(* CODESYS project FanucSimpleLibrary.library
   Author: Yonatan Avrakh
   Version: 0.1.0.0
   Description: A simple library allowing fast integration with FANUC robot
   Title: FanucSimple
   DefaultNamespace: FanucSimple
   Placeholder: FanucSimple
   Company: Beckhoff Automation IL

Project tree, tasks and I/O mapping:
  libraries: Tc2_Standard, * (Beckhoff Automation GmbH); Tc2_System, * (Beckhoff Automation GmbH)
  DUTs/
    data type E_FanucCstopiState
    data type E_FanucEnableState
    data type E_FanucFaultResetState
    data type E_FanucHomingState
    data type E_FanucStartProgramState
    data type ST_FanucControl
    data type ST_FanucStatus
  GVLs/
  POUs/
    function block FB_FanucControl [ST]
    function block FB_FanucCycleStop [ST]
    function block FB_FanucEnable [ST]
    function block FB_FanucFaultReset [ST]
    function block FB_FanucHoming [ST]
    function block FB_FanucOverwrite [ST]
    function block FB_FanucStartProgram [ST]
    function block FB_FanucStatus [ST]
  Version/
    global variables Global_Version
  VISUs/
*)

// DUTs/E_FanucCstopiState
(*
  States for FB_FanucCycleStop.
  Sequence: Idle → Pulsing → Done (→ Idle)
*)
TYPE E_FanucCstopiState :
(
	Idle    := 0,   // Waiting for bTrigger rising edge.
	Pulsing := 1,   // CSTOPI signal pulsed for 20 ms.
	Done    := 2    // Cycle stop complete – bDone TRUE for one scan, then → Idle.
);
END_TYPE

// DUTs/E_FanucEnableState
(*
  States for FB_FanucEnable.
  The enable sequence progresses: Idle → ClearFault → CheckTP → WaitReady → Ready.
  From Ready, conditions are monitored continuously (priority order):
    bFault             → ClearFault
    bTP_Enabled        → CheckTP
    bExtIMSTP = FALSE  → EmergencyStop (E-stop; resumes via ClearFault when released)
    bExtSFSPD = FALSE  → SafeSpeed     (fence open; robot at safe speed; bReady FALSE)
    bExtHold  = FALSE  → Paused        (HOLD only drops; IMSTP/SFSPD/ENBL held)
  Toggle bEnable FALSE→TRUE to retry from Idle after an Error.
*)
TYPE E_FanucEnableState :
(
  Idle              := 0,   // Waiting for bEnable. ENBL de-asserted; bExt* signals pass through.
  ClearFault        := 1,   // Assert Fault_Reset pulse until bFault clears (5 s timeout → Error).
  CheckTP           := 3,   // Wait for bTP_Enabled = FALSE (operator must switch TP off).
  WaitReady         := 4,   // Wait for bCmd_Enabled AND bSystem_Ready (5 s timeout → Error).
  Ready             := 5,   // Robot is ready. Monitor for all safety/fault conditions.
  Paused            := 6,   // bExtHold = FALSE: HOLD dropped, IMSTP/SFSPD/ENBL held. Resumes when bExtHold TRUE.
  EmergencyStop     := 7,   // bExtIMSTP = FALSE: E-stop active. ENBL held. Resumes via ClearFault when IMSTP released.
  SafeSpeed         := 8,   // bExtSFSPD = FALSE: fence open, robot at safe speed. bReady FALSE. Resumes when fence closes.
  Error             := 99   // Enable sequence failed. ENBL de-asserted. Toggle bEnable to reset.
);
END_TYPE

// DUTs/E_FanucFaultResetState
(*
  States for FB_FanucFaultReset.
  Sequence: Idle → SendPulse → WaitClear → Done (→ Idle).
  Error on timeout; reset by setting bReset FALSE.
*)
TYPE E_FanucFaultResetState :
(
  Idle      := 0,   // Waiting for bReset rising edge.
  SendPulse := 1,   // FAULT_RESET signal pulsed for 20 ms (robot acts on rising edge).
  WaitClear := 2,   // Waiting for bFault = FALSE (configurable timeout → Error).
  Done      := 3,   // Fault cleared – bDone TRUE for one scan, then → Idle.
  Error     := 99   // Fault persisted after reset attempt. Set bReset FALSE to reset.
);
END_TYPE

// DUTs/E_FanucHomingState
(*
  States for FB_FanucHoming.
  Sequence: Idle → RequestHome → WaitComplete → Done (→ Idle).
  Error on timeout; reset by setting bStart FALSE.
*)
TYPE E_FanucHomingState :
(
  Idle         := 0,   // Waiting for bStart rising edge (interlocked by bReady).
  RequestHome  := 1,   // HOME signal (UI[7]) pulsed for 20 ms to trigger homing macro.
  WaitComplete := 2,   // Waiting for bAt_Home (UO[7]) = TRUE (configurable timeout).
  Done         := 3,   // Homing confirmed – bDone TRUE for one scan, then → Idle.
  Error        := 99   // Timeout waiting for completion. Set bStart FALSE to reset.
);
END_TYPE

// DUTs/E_FanucStartProgramState
(*
  States for FB_FanucStartProgram.
  Sequence: Idle → Pulsing → Done (→ Idle)
  Error on invalid program number; reset by setting bStart FALSE.
*)
TYPE E_FanucStartProgramState :
(
	Idle    := 0,   // Waiting for bStart rising edge.
	Pulsing := 1,   // Program start bits asserted for 200 ms.
	Done    := 2,   // Pulse complete – bDone TRUE for one scan, then → Idle.
	Error   := 99   // Program number out of range. Set bStart FALSE to reset.
);
END_TYPE

// DUTs/ST_FanucControl
TYPE ST_FanucControl : STRUCT
//  Control byte 0
  IMSTP        :  BOOL;  //  (* bit 0 *)
  Hold        :  BOOL;  //  (* bit 1 *)
  SFSPD        :  BOOL;  //  (* bit 2 *)
  Cycle_stop      :  BOOL;  //  (* bit 3 *)
  Fault_Reset      :  BOOL;  //  (* bit 4 *)
  Start        :  BOOL;  //  (* bit 5 *)
  Home        :  BOOL;  //  (* bit 6 *)
  Enable        :  BOOL;  //  (* bit 7 *)

//  Control byte 1  (UI[9..16]  RSR1..RSR8 / PNS1..PNS8)
  Start_Program1    :  BOOL;  //  UI[9]  RSR1 / PNS bit 0
  Start_Program2    :  BOOL;  //  UI[10] RSR2 / PNS bit 1
  Start_Program3    :  BOOL;  //  UI[11] RSR3 / PNS bit 2
  Start_Program4    :  BOOL;  //  UI[12] RSR4 / PNS bit 3
  Start_Program5    :  BOOL;  //  UI[13] RSR5 / PNS bit 4
  Start_Program6    :  BOOL;  //  UI[14] RSR6 / PNS bit 5
  Start_Program7    :  BOOL;  //  UI[15] RSR7 / PNS bit 6
  Start_Program8    :  BOOL;  //  UI[16] RSR8 / PNS bit 7

//  Control byte 2  (UI[17..18])
  PNS_Strobe      :  BOOL;
  Prod_Start      :  BOOL;  //  UI[18] PROD_START – triggers PNS program execution

//  Control byte 3  (GI[25..33] – user-defined output)
  Overwrite            :  BYTE;
END_STRUCT
END_TYPE

// DUTs/ST_FanucStatus
TYPE ST_FanucStatus : STRUCT
  //DI[0,0] - Status Byte 0
  bCmd_Enabled  : BOOL;  (* bit 0 *)
  bSystem_Ready  : BOOL;  (* bit 1 *)
  bPrg_Running  : BOOL;  (* bit 2 *)
  bPrg_Paused    : BOOL;  (* bit 3 *)
  bMotion_Held  : BOOL;  (* bit 4 *)
  bFault      : BOOL;  (* bit 5 *)
  bAt_Home    : BOOL;  (* bit 6 *)
  bTP_Enabled    : BOOL;  (* BIT 7 *)

  //DI[0,1] - Status Byte 1
  bBatteryAlarm :BOOL; (* bit 1 *)
  bBusy :BOOL;  (* bit 2 *)

  //DI[0,2] - Status Byte 2
  bProg_Start1ACK  : BOOL;  (* bit 1 *)
  bProg_Start2ACK  : BOOL;  (* bit 2 *)
  bProg_Start3ACK  : BOOL;  (* bit 3 *)
  bProg_Start4ACK  : BOOL;  (* bit 4 *)
  bProg_Start5ACK  : BOOL;  (* bit 5 *)
  bProg_Start6ACK  : BOOL;  (* bit 6 *)
  bProg_Start7ACK  : BOOL;  (* bit 7 *)
  bProg_Start8ACK  : BOOL;  (* bit 8 *)

END_STRUCT
END_TYPE

// Version/Global_Version
{attribute 'TcGenerated'}
{attribute 'no-analysis'}
{attribute 'linkalways'}
// This function has been automatically generated from the project information.
VAR_GLOBAL CONSTANT
	{attribute 'const_non_replaced'}
	stLibVersion_FanucSimple : ST_LibVersion := (iMajor := 0, iMinor := 1, iBuild := 0, iRevision := 0, nFlags := 1, sVersion := '0.1.0.0');
END_VAR

// POUs/FB_FanucControl
(* Writes ST_FanucControl fields TO EtherCAT output bytes (aDO). Call every scan AFTER all control logic is complete. Pass GVL_Fanuc.DO0 AT the call site
*)
FUNCTION_BLOCK FB_FanucControl
VAR_IN_OUT
  aDO : ARRAY[0..15] OF BYTE; // Injected EtherCAT output array – pass GVL_Fanuc.DO0
END_VAR
VAR_INPUT
  stControl : ST_FanucControl;
END_VAR


// Control Byte 0  (aDO[0])  —  UI[1..8]
aDO[0].0 := stControl.IMSTP;        // UI[1]  *IMSTP       NC – hold TRUE; FALSE = software E-stop
aDO[0].1 := stControl.Hold;         // UI[2]  *HOLD        NC – hold TRUE; FALSE = decelerate & pause
aDO[0].2 := stControl.SFSPD;        // UI[3]  *SFSPD       NC – hold TRUE; FALSE = safe-speed limit
aDO[0].3 := stControl.Cycle_stop;   // UI[4]  CSTOPI       pulse to stop/abort current cycle
aDO[0].4 := stControl.Fault_Reset;  // UI[5]  FAULT_RESET  pulse to reset clearable alarms
aDO[0].5 := stControl.Start;        // UI[6]  START        falling-edge resumes paused program
aDO[0].6 := stControl.Home;         // UI[7]  HOME         macro use only
aDO[0].7 := stControl.Enable;       // UI[8]  ENBL         NC – hold TRUE; FALSE = disable all motion

// Control Byte 1  (aDO[1])  —  UI[9..16]  RSR / PNS
aDO[1].0 := stControl.Start_Program1; // UI[9]  RSR1 / PNS bit 0
aDO[1].1 := stControl.Start_Program2; // UI[10] RSR2 / PNS bit 1
aDO[1].2 := stControl.Start_Program3; // UI[11] RSR3 / PNS bit 2
aDO[1].3 := stControl.Start_Program4; // UI[12] RSR4 / PNS bit 3
aDO[1].4 := stControl.Start_Program5; // UI[13] RSR5 / PNS bit 4
aDO[1].5 := stControl.Start_Program6; // UI[14] RSR6 / PNS bit 5
aDO[1].6 := stControl.Start_Program7; // UI[15] RSR7 / PNS bit 6
aDO[1].7 := stControl.Start_Program8; // UI[16] RSR8 / PNS bit 7

// Control Byte 2  (aDO[2])  —  UI[17..18]
aDO[2].0 := stControl.PNS_Strobe;                   // UI[17] reserved
aDO[2].1 := stControl.Prod_Start;   // UI[18] PROD_START – triggers PNS program execution

// Control Byte 3  (aDO[3])  —  GI[25..33] user-defined output
aDO[3] := stControl.Overwrite;

END_FUNCTION_BLOCK

// POUs/FB_FanucCycleStop
// Sends the CSTOPI (UI[4]) Cycle Stop signal to the FANUC robot.
// Rising edge on bTrigger sends a 20 ms pulse; bDone goes TRUE for one scan when complete.
FUNCTION_BLOCK FB_FanucCycleStop
VAR_INPUT
  bTrigger   : BOOL;   // Rising edge: send Cycle Stop command
END_VAR
VAR_IN_OUT
  stControl  : ST_FanucControl;   // Control struct – wire same instance as FB_FanucEnable output
END_VAR
VAR_OUTPUT
  bBusy      : BOOL;               // TRUE while pulse is active
  bDone      : BOOL;               // One scan TRUE when cycle stop pulse is complete
  eState     : E_FanucCstopiState; // Current state (diagnostic / HMI)
END_VAR
VAR
  _eState   : E_FanucCstopiState := E_FanucCstopiState.Idle;
  rtTrigger : R_TRIG;
  tonPulse  : TON;   // 20 ms CSTOPI pulse width
END_VAR
VAR CONSTANT
  tPulse : TIME := T#20MS;   // CSTOPI minimum pulse width (spec: ≥15 ms)
END_VAR

(*
  FB_FanucCycleStop
  Sends a 20 ms CSTOPI pulse (UI[4]) to the FANUC robot.

  CSTOPI clears programs waiting on RSR. The effect on the running program depends
  on the "CSTOPI for ABORT" setting on the controller (MENU → SYSTEM → Config item 6):
    DISABLE – program stops at the end of its current cycle (graceful stop).
    ENABLE  – program is immediately aborted at the current line.
  This FB sends the pulse unconditionally; the controller setting determines the behaviour.

  Usage:
    - Call every PLC cycle.
    - Pass the same stControl instance used by FB_FanucEnable and FB_FanucControl.
    - Give bTrigger a rising edge to issue the command.
    - bDone goes TRUE for one scan when the 20 ms pulse is complete.
*)

// ---------- Edge detect ----------
rtTrigger(CLK := bTrigger);

// ---------- State machine ----------
CASE _eState OF

  E_FanucCstopiState.Idle:
    stControl.Cycle_stop := FALSE;
    tonPulse(IN := FALSE);
    IF rtTrigger.Q THEN
      _eState := E_FanucCstopiState.Pulsing;
    END_IF

  E_FanucCstopiState.Pulsing:
    // Assert CSTOPI for 20 ms, then → Done.
    tonPulse(IN := TRUE, PT := tPulse);
    stControl.Cycle_stop := NOT tonPulse.Q;  // TRUE for first 20 ms, then FALSE
    IF tonPulse.Q THEN
      stControl.Cycle_stop := FALSE;
      tonPulse(IN := FALSE);
      _eState := E_FanucCstopiState.Done;
    END_IF

  E_FanucCstopiState.Done:
    // bDone is TRUE for one scan (derived below), then → Idle.
    stControl.Cycle_stop := FALSE;
    _eState := E_FanucCstopiState.Idle;

ELSE
  _eState := E_FanucCstopiState.Idle;

END_CASE

// ---------- Derived outputs ----------
eState := _eState;
bBusy  := (_eState = E_FanucCstopiState.Pulsing);
bDone  := (_eState = E_FanucCstopiState.Done);

END_FUNCTION_BLOCK

// POUs/FB_FanucEnable
// Runs the FANUC enable sequence (IMSTP/HOLD/SFSPD → ClearFault → CheckTP → WaitReady → Ready).
// Validates interlock preconditions before enabling. Set bEnable TRUE to start; toggle FALSE→TRUE to reset after error.
FUNCTION_BLOCK FB_FanucEnable
VAR_INPUT
  bEnable    : BOOL;           // Command: TRUE to run enable sequence
  stStatus   : ST_FanucStatus; // Live robot status (from FB_FanucStatus)
  // External interlock signals – Normally Closed convention: TRUE = normal, FALSE = activate stop/hold
  // May be driven by HMI, safety PLC, or TwinCAT logic. Merged at the call site; this FB sees one value per signal.
  bExtIMSTP  : BOOL;  // External *IMSTP: FALSE = E-stop requested
  bExtHold   : BOOL;  // External *HOLD:  FALSE = pause/hold requested
  bExtSFSPD  : BOOL;  // External *SFSPD: FALSE = safe-speed limit requested
  bExtStart  : BOOL;  // External Start command: rising edge triggers a 20 ms START pulse (Ready state only)
END_VAR
VAR_OUTPUT
  bReady          : BOOL;                // Robot is ready to execute programs
  bError          : BOOL;                // Enable sequence failed – check eState
  bTPWarning      : BOOL;                // TP switch is ON – operator action needed
  eState          : E_FanucEnableState;  // Current state (diagnostic / HMI)
  stControl       : ST_FanucControl;     // Control outputs – wire to FB_FanucControl
END_VAR
VAR
  _eState          : E_FanucEnableState := E_FanucEnableState.Idle;
  tonReadyTimeout  : TON;   // Timeout waiting for CMDENBL + SYSRDY (5 s → Error)
  rtExtStart       : R_TRIG;  // Rising-edge detector for bExtStart
  tonStartPulse    : TON;   // 20 ms START pulse generator
END_VAR
VAR CONSTANT
  tStartPulse : TIME := T#20MS;  // START signal minimum pulse width
END_VAR

(*
  FB_FanucEnable
  Implements the FANUC robot enable sequence as a state machine.

  Sequence (per FANUC UI/UO signal spec):
    0. Idle       – bEnable must be TRUE and all interlocks in required state before proceeding.
    1. ClearFault – Waits for bFault = FALSE. Does NOT send a reset pulse; use FB_FanucFaultReset.
    2. CheckTP    – Wait for bTP_Enabled = FALSE. TP switch must be OFF for remote control.
    3. WaitReady  – Wait for bCmd_Enabled AND bSystem_Ready (5 s timeout → Error).
    4. Ready      – bReady = TRUE. Continuously monitors for fault/TP/hold/interlock changes.

  To reset after Error: set bEnable FALSE, then TRUE again.

  Fault clearing:
    This FB does not send FAULT_RESET. When in ClearFault state, call FB_FanucFaultReset
    (passing the same stControl instance) and trigger it with bReset. FB_FanucEnable will
    transition out of ClearFault automatically once bFault = FALSE.

  NC signal behaviour (Option A – passive when disabled):
    When bEnable = FALSE (Idle or Error): IMSTP, HOLD, SFSPD are held TRUE (non-asserting).
    ENBL = FALSE is the primary gate; additional stop assertions would cause unnecessary alarms.
    When in any active state: NC signals reflect bExt* inputs directly.

  Emergency Stop (bExtIMSTP = FALSE from Ready/Paused/SafeSpeed):
    → EmergencyStop. NC signal drops immediately; robot stops. ENBL stays asserted for recovery.
    No fault-clear while IMSTP is low. When bExtIMSTP returns TRUE → ClearFault.

  Safe Speed (bExtSFSPD = FALSE from Ready/Paused):
    → SafeSpeed. Robot continues at safe speed; bReady = FALSE.
    When bExtSFSPD returns TRUE: → Ready (if bExtHold TRUE) or → Paused.

  Pause / Hold (bExtHold = FALSE from Ready):
    → Paused. Only HOLD is dropped; IMSTP, SFSPD and ENBL remain asserted.
    When bExtHold returns TRUE → Ready.

  Start (bExtStart):
    Rising edge in Ready state triggers a 20 ms pulse on stControl.Start (UI[6]).
    Must be FALSE before the enable sequence can begin.

  Library usage:
    - Call every PLC cycle.
    - Pass fbStatus.stStatus into stStatus.
    - Wire stControl output to FB_FanucControl (inject aDO at call site).
    - Program start, homing, and cycle-stop bits are not managed here;
      handle those in the calling application or a dedicated FB.
*)

// ------------------- NC safety signals — always reflect external inputs directly -------------------
stControl.IMSTP := bExtIMSTP;
stControl.Hold  := bExtHold;
stControl.SFSPD := bExtSFSPD;

// ------------------- State machine – transition logic only -------------------
CASE _eState OF

  E_FanucEnableState.Idle:
    tonReadyTimeout(IN := FALSE);
    // All interlock preconditions must be met before starting the enable sequence.
    IF bEnable AND bExtIMSTP AND bExtHold AND bExtSFSPD AND NOT bExtStart THEN
      _eState := E_FanucEnableState.ClearFault;
    END_IF

  E_FanucEnableState.ClearFault:
    // Wait for bFault to clear. No pulse is sent here – use FB_FanucFaultReset for that.
    // Abort back to Idle if bEnable dropped or any interlock was lost mid-sequence.
    IF NOT bEnable OR NOT bExtIMSTP OR NOT bExtHold OR NOT bExtSFSPD THEN
      _eState := E_FanucEnableState.Idle;
    ELSIF NOT stStatus.bFault THEN
      _eState := E_FanucEnableState.CheckTP;
    END_IF

  E_FanucEnableState.CheckTP:
    // bTPWarning is derived below; stay here until operator switches TP off.
    // Abort if bEnable dropped or any interlock was lost mid-sequence.
    IF NOT bEnable OR NOT bExtIMSTP OR NOT bExtHold OR NOT bExtSFSPD THEN
      _eState := E_FanucEnableState.Idle;
    ELSIF NOT stStatus.bTP_Enabled THEN
      tonReadyTimeout(IN := FALSE);
      _eState := E_FanucEnableState.WaitReady;
    END_IF

  E_FanucEnableState.WaitReady:
    // Wait for CMDENBL (UO1) and SYSRDY (UO2) to confirm the robot is ready.
    // Interlock loss takes highest priority – abort cleanly rather than time out.
    tonReadyTimeout(IN := TRUE, PT := T#5S);
    IF NOT bEnable OR NOT bExtIMSTP OR NOT bExtHold OR NOT bExtSFSPD THEN
      tonReadyTimeout(IN := FALSE);
      _eState := E_FanucEnableState.Idle;
    ELSIF stStatus.bCmd_Enabled AND stStatus.bSystem_Ready THEN
      tonReadyTimeout(IN := FALSE);
      _eState := E_FanucEnableState.Ready;
    ELSIF stStatus.bTP_Enabled THEN
      tonReadyTimeout(IN := FALSE);
      _eState := E_FanucEnableState.CheckTP;
    ELSIF stStatus.bFault THEN
      tonReadyTimeout(IN := FALSE);
      _eState := E_FanucEnableState.ClearFault;
    ELSIF tonReadyTimeout.Q THEN
      _eState := E_FanucEnableState.Error;
    END_IF

  E_FanucEnableState.Ready:
    // Monitor all conditions (priority: fault > TP > E-stop > SafeSpeed > Hold).
    IF NOT bEnable THEN
      _eState := E_FanucEnableState.Idle;
    ELSIF stStatus.bFault THEN
      _eState := E_FanucEnableState.ClearFault;
    ELSIF stStatus.bTP_Enabled THEN
      _eState := E_FanucEnableState.CheckTP;
    ELSIF NOT bExtIMSTP THEN
      _eState := E_FanucEnableState.EmergencyStop;
    ELSIF NOT bExtSFSPD THEN
      _eState := E_FanucEnableState.SafeSpeed;
    ELSIF stStatus.bMotion_Held THEN
      _eState := E_FanucEnableState.Paused;
    END_IF

  E_FanucEnableState.Paused:
    // HOLD NC already low via passthrough. ENBL remains asserted.
    IF NOT bEnable THEN
      _eState := E_FanucEnableState.Idle;
    ELSIF stStatus.bFault THEN
      _eState := E_FanucEnableState.ClearFault;
    ELSIF stStatus.bTP_Enabled THEN
      _eState := E_FanucEnableState.CheckTP;
    ELSIF NOT bExtIMSTP THEN
      _eState := E_FanucEnableState.EmergencyStop;
    ELSIF NOT bExtSFSPD THEN
      _eState := E_FanucEnableState.SafeSpeed;
    ELSIF NOT stStatus.bMotion_Held THEN
      _eState := E_FanucEnableState.Ready;
    END_IF

  E_FanucEnableState.EmergencyStop:
    // IMSTP NC already low via passthrough. ENBL stays asserted for recovery.
    // Do NOT attempt fault-clear while IMSTP is still low.
    IF NOT bEnable THEN
      _eState := E_FanucEnableState.Idle;
    ELSIF stStatus.bTP_Enabled THEN
      _eState := E_FanucEnableState.CheckTP;
    ELSIF bExtIMSTP THEN
      // E-stop released – robot almost certainly alarmed; pass through ClearFault.
      _eState := E_FanucEnableState.ClearFault;
    END_IF

  E_FanucEnableState.SafeSpeed:
    // SFSPD NC already low via passthrough; robot runs at safe speed.
    IF NOT bEnable THEN
      _eState := E_FanucEnableState.Idle;
    ELSIF stStatus.bFault THEN
      _eState := E_FanucEnableState.ClearFault;
    ELSIF stStatus.bTP_Enabled THEN
      _eState := E_FanucEnableState.CheckTP;
    ELSIF NOT bExtIMSTP THEN
      _eState := E_FanucEnableState.EmergencyStop;
    ELSIF bExtSFSPD THEN
      // Fence closed – resume; honour hold state.
      IF bExtHold THEN
        _eState := E_FanucEnableState.Ready;
      ELSE
        _eState := E_FanucEnableState.Paused;
      END_IF
    END_IF

  E_FanucEnableState.Error:
    // ENBL de-asserted (derived below). Reset by toggling bEnable FALSE → TRUE.
    IF NOT bEnable THEN
      tonReadyTimeout(IN := FALSE);
      _eState := E_FanucEnableState.Idle;
    END_IF

ELSE
  _eState := E_FanucEnableState.Error;

END_CASE

//-------------------START pulse-------------------
//  Convert rising edge of bExtStart into a clean 20 ms pulse on stControl.Start.
//  Gated by Ready state – rising edges in any other state are ignored.
//  If we leave Ready mid-pulse (e.g. fault occurs), the timer resets cleanly. *)
rtExtStart(CLK := bExtStart AND (_eState = E_FanucEnableState.Ready));
tonStartPulse(IN := tonStartPulse.IN OR rtExtStart.Q, PT := tStartPulse);
IF tonStartPulse.Q THEN
  tonStartPulse(IN := FALSE);
END_IF
IF _eState <> E_FanucEnableState.Ready THEN
  tonStartPulse(IN := FALSE);
END_IF

// -------------------Derived outputs-------------------
// Evaluated after the state machine so they always reflect the current state. *)
eState             := _eState;
stControl.Enable   := (_eState <> E_FanucEnableState.Idle)  AND (_eState <> E_FanucEnableState.Error);
stControl.Start    := (_eState =  E_FanucEnableState.Ready) AND tonStartPulse.IN;
bReady             := (_eState =  E_FanucEnableState.Ready);
bError             := (_eState =  E_FanucEnableState.Error);
bTPWarning         := (_eState =  E_FanucEnableState.CheckTP) AND stStatus.bTP_Enabled;

END_FUNCTION_BLOCK

// POUs/FB_FanucFaultReset
// Sends a FAULT_RESET pulse to the FANUC robot and waits for the fault to clear.
// Trigger with a rising edge on bReset. Toggle bReset FALSE to reset after Error.
FUNCTION_BLOCK FB_FanucFaultReset
VAR_INPUT
  bReset   : BOOL;            // Rising edge: send fault reset pulse to robot
  stStatus : ST_FanucStatus;  // Live robot status (from FB_FanucStatus)
END_VAR
VAR_IN_OUT
  stControl : ST_FanucControl;  // Control struct – pass same instance as FB_FanucEnable.stControl
END_VAR
VAR_OUTPUT
  bBusy  : BOOL;                    // TRUE while reset sequence is in progress
  bDone  : BOOL;                    // One scan TRUE when fault is confirmed cleared
  bError : BOOL;                    // Fault persisted after reset – operator action needed
  eState : E_FanucFaultResetState;  // Current state (diagnostic / HMI)
END_VAR
VAR
  _eState    : E_FanucFaultResetState := E_FanucFaultResetState.Idle;
  rtReset    : R_TRIG;
  tonPulse   : TON;  // 20 ms FAULT_RESET pulse
  tonTimeout : TON;  // Timeout waiting for fault to clear after reset
END_VAR
VAR CONSTANT
  tResetPulse   : TIME := T#20MS;  // FAULT_RESET minimum pulse width
  tFaultTimeout : TIME := T#5S;    // Max time to wait for fault to clear after reset
END_VAR

(*
  FB_FanucFaultReset
  Sends a timed FAULT_RESET pulse (UI[5]) to the robot and monitors bFault until clear.

  Sequence:
    1. SendPulse  – Assert FAULT_RESET for 20 ms. Robot acts on the rising edge.
    2. WaitClear  – Wait for bFault (UO[4]) = FALSE. Timeout → Error.
    3. Done       – bDone TRUE for one scan, then → Idle.

  Usage:
    - Call every PLC cycle.
    - Pass the same stControl instance used by FB_FanucEnable (VAR_IN_OUT, by reference).
    - Trigger with a rising edge on bReset (e.g. HMI button, or automatic from application logic).
    - Check bDone for one-scan confirmation that the fault cleared.
    - Check bError if the fault did not clear; set bReset FALSE to reset.

  Relationship with FB_FanucEnable:
    - FB_FanucEnable.ClearFault state waits for bFault = FALSE without sending any pulse.
    - This FB is responsible for the actual reset signal; the application decides when to trigger it.
    - Typically called when FB_FanucEnable.eState = ClearFault and the operator requests a reset.
*)

rtReset(CLK := bReset);

CASE _eState OF

  E_FanucFaultResetState.Idle:
    stControl.Fault_Reset := FALSE;
    tonPulse(IN := FALSE);
    tonTimeout(IN := FALSE);
    IF rtReset.Q THEN
      _eState := E_FanucFaultResetState.SendPulse;
    END_IF

  E_FanucFaultResetState.SendPulse:
    // Assert FAULT_RESET for exactly 20 ms. Robot acts on the rising edge.
    tonPulse(IN := TRUE, PT := tResetPulse);
    stControl.Fault_Reset := NOT tonPulse.Q; // TRUE for first 20 ms, then FALSE
    IF tonPulse.Q THEN
      stControl.Fault_Reset := FALSE;
      tonPulse(IN := FALSE);
      _eState := E_FanucFaultResetState.WaitClear;
    END_IF

  E_FanucFaultResetState.WaitClear:
    // Pulse complete; wait for robot to confirm the fault is gone.
    stControl.Fault_Reset := FALSE;
    tonTimeout(IN := TRUE, PT := tFaultTimeout);
    IF NOT stStatus.bFault THEN
      tonTimeout(IN := FALSE);
      _eState := E_FanucFaultResetState.Done;
    ELSIF tonTimeout.Q THEN
      _eState := E_FanucFaultResetState.Error;
    END_IF

  E_FanucFaultResetState.Done:
    // bDone is TRUE for exactly one scan (derived below), then return to Idle.
    stControl.Fault_Reset := FALSE;
    _eState := E_FanucFaultResetState.Idle;

  E_FanucFaultResetState.Error:
    // Fault did not clear after reset. Reset this FB by setting bReset FALSE.
    stControl.Fault_Reset := FALSE;
    IF NOT bReset THEN
      tonPulse(IN := FALSE);
      tonTimeout(IN := FALSE);
      _eState := E_FanucFaultResetState.Idle;
    END_IF

ELSE
  _eState := E_FanucFaultResetState.Error;

END_CASE

// ---------- Derived outputs ---------- *)
eState := _eState;
bBusy  := (_eState = E_FanucFaultResetState.SendPulse) OR (_eState = E_FanucFaultResetState.WaitClear);
bDone  := (_eState = E_FanucFaultResetState.Done);
bError := (_eState = E_FanucFaultResetState.Error);

END_FUNCTION_BLOCK

// POUs/FB_FanucStatus
//Reads EtherCAT input bytes (aDI) into ST_FanucStatus. Call every scan BEFORE any status-dependent logic. Pass GVL_Fanuc.DI0 at the call site.
FUNCTION_BLOCK FB_FanucStatus
VAR_IN_OUT
  aDI : ARRAY[0..15] OF BYTE; // Injected EtherCAT input array – pass GVL_Fanuc.DI0
END_VAR
VAR_OUTPUT
  stStatus : ST_FanucStatus;
END_VAR

(*
  FB_FanucStatus
  Reads the raw EtherCAT input byte array (injected as aDI) and maps
  each bit to the corresponding field in ST_FanucStatus.

  Call every PLC cycle BEFORE any logic that depends on robot status.

  Library usage – I/O injection:
    The caller passes the hardware-linked byte array at the call site:
      fbStatus(aDI := GVL_Fanuc.DI0, stStatus => stStatus);
    This keeps AT %I* declarations out of the library.

  Signal mapping (FANUC R-30iB Plus, PDO3 – Receive PDO3):
    aDI[0]  ← Robot UO[1..8]   (CMDENBL, SYSRDY, PROGRUN, PAUSED, HELD, FAULT, ATPERCH, TPENBL)
    aDI[1]  ← Robot UO[9..10]  (BATALM, BUSY)
    aDI[2]  ← Robot UO[11..18] (ACK1..ACK8 / SNO1..SNO8)
*)


// Status Byte 0  (aDI[0])  —  UO[1..8]
stStatus.bCmd_Enabled  := aDI[0].0;   // UO[1]  CMDENBL  – command enable
stStatus.bSystem_Ready := aDI[0].1;   // UO[2]  SYSRDY   – servo powered, no alarm
stStatus.bPrg_Running  := aDI[0].2;   // UO[3]  PROGRUN  – program in execution
stStatus.bPrg_Paused   := aDI[0].3;   // UO[4]  PAUSED   – program on hold
stStatus.bMotion_Held  := aDI[0].4;   // UO[5]  HELD     – HOLD button/signal active
stStatus.bFault        := aDI[0].5;   // UO[6]  FAULT    – alarm preventing execution
stStatus.bAt_Home      := aDI[0].6;   // UO[7]  ATPERCH  – robot at reference position 1
stStatus.bTP_Enabled   := aDI[0].7;   // UO[8]  TPENBL   – teach pendant enable switch ON

// Status Byte 1  (aDI[1])  —  UO[9..10]
stStatus.bBatteryAlarm := aDI[1].0;   // UO[9]  BATALM   – controller battery low
stStatus.bBusy         := aDI[1].1;   // UO[10] BUSY     – program executing or TP busy

// Status Byte 2  (aDI[2])  —  UO[11..18]  RSR ACK / SNO
stStatus.bProg_Start1ACK := aDI[2].0; // UO[11] ACK1/SNO1
stStatus.bProg_Start2ACK := aDI[2].1; // UO[12] ACK2/SNO2
stStatus.bProg_Start3ACK := aDI[2].2; // UO[13] ACK3/SNO3
stStatus.bProg_Start4ACK := aDI[2].3; // UO[14] ACK4/SNO4
stStatus.bProg_Start5ACK := aDI[2].4; // UO[15] ACK5/SNO5
stStatus.bProg_Start6ACK := aDI[2].5; // UO[16] ACK6/SNO6
stStatus.bProg_Start7ACK := aDI[2].6; // UO[17] ACK7/SNO7
stStatus.bProg_Start8ACK := aDI[2].7; // UO[18] ACK8/SNO8

END_FUNCTION_BLOCK

// POUs/FB_FanucHoming
// Executes the FANUC robot homing sequence via HOME (UI[7]).
// Rising edge on bStart triggers a 20 ms HOME pulse to call the homing macro on the robot.
// Completion is confirmed by bAt_Home (UO[7]) going TRUE. Set bStart FALSE to reset after Error.
FUNCTION_BLOCK FB_FanucHoming
VAR_INPUT
  bStart    : BOOL;            // Rising edge: start homing (interlocked by bReady)
  bReady    : BOOL;            // From FB_FanucEnable.bReady – homing only starts when robot is enabled
  stStatus  : ST_FanucStatus;  // Live robot status
END_VAR
VAR_IN_OUT
  stControl : ST_FanucControl; // Control struct – wire same instance as FB_FanucEnable output
END_VAR
VAR_OUTPUT
  bBusy     : BOOL;                 // TRUE while homing is in progress
  bDone     : BOOL;                 // One scan TRUE when bAt_Home confirmed
  bError    : BOOL;                 // TRUE on timeout; set bStart FALSE to reset
  eState    : E_FanucHomingState;   // Current state (diagnostic / HMI)
END_VAR
VAR
  _eState         : E_FanucHomingState := E_FanucHomingState.Idle;
  rtStart         : R_TRIG;
  tonHomePulse    : TON;   // 20 ms HOME signal pulse
  tonWaitComplete : TON;   // Timeout waiting for bAt_Home (configurable via tHomingTimeout)
END_VAR
VAR CONSTANT
  tHomePulse    : TIME := T#200MS;  // HOME signal minimum pulse width
  tHomingTimeout : TIME := T#30S; // Max time allowed for homing macro to complete
END_VAR

(*
  FB_FanucHoming
  Executes the robot homing procedure as a state machine.

  HOME (UI[7]) is configured on the FANUC controller to trigger a macro (typically a Karel
  or TP program) that drives the robot to its home position.  Completion is indicated by
  bAt_Home (UO[7]) going TRUE.

  Sequence:
    1. RequestHome  – Assert HOME (UI[7]) for 20 ms to trigger the homing macro.
    2. WaitComplete – Wait for bAt_Home (UO[7]) = TRUE (timeout: tHomingTimeout).
    3. Done         – bDone TRUE for one scan; state returns to Idle.

  Interlocks:
    - bStart is edge-detected and gated by bReady. Homing is only triggered when the
      robot is enabled and ready for remote operation.
    - If bAt_Home is already TRUE when homing is requested, WaitComplete completes
      immediately and bDone is asserted for one scan.

  Error handling:
    - If bAt_Home does not go TRUE within tHomingTimeout, the FB transitions to Error.
    - Set bStart FALSE to acknowledge and reset to Idle.

  Prerequisites on the FANUC controller:
    - A macro or TP program must be assigned to the HOME input (UI[7]).
    - UO[7] (At Perch/Home) must be configured to reflect the robot's home position.

  Usage:
    - Call every PLC cycle.
    - Pass the same stControl instance used by FB_FanucEnable and FB_FanucControl.
    - Wire bReady from FB_FanucEnable.bReady.
    - Give bStart a rising edge to begin. Monitor bBusy / bDone / bError.
*)

// ---------- Edge detect ----------
rtStart(CLK := bStart AND bReady);

// ---------- State machine ----------
CASE _eState OF

  E_FanucHomingState.Idle:
    stControl.Home := FALSE;
    tonHomePulse(IN := FALSE);
    tonWaitComplete(IN := FALSE);
    IF rtStart.Q THEN
      _eState := E_FanucHomingState.RequestHome;
    END_IF

  E_FanucHomingState.RequestHome:
    // Assert HOME (UI[7]) for 20 ms to trigger the homing macro.
    tonHomePulse(IN := TRUE, PT := tHomePulse);
    stControl.Home := NOT tonHomePulse.Q;  // TRUE for first 20 ms, then FALSE
    IF tonHomePulse.Q THEN
      stControl.Home := FALSE;
      tonHomePulse(IN := FALSE);
      _eState := E_FanucHomingState.WaitComplete;
    END_IF

  E_FanucHomingState.WaitComplete:
    // Wait for the robot to confirm it has reached home (UO[7]).
    // If bAt_Home is already TRUE the state completes immediately.
    stControl.Home := FALSE;
    tonWaitComplete(IN := TRUE, PT := tHomingTimeout);
    IF stStatus.bAt_Home THEN
      tonWaitComplete(IN := FALSE);
      _eState := E_FanucHomingState.Done;
    ELSIF tonWaitComplete.Q THEN
      tonWaitComplete(IN := FALSE);
      _eState := E_FanucHomingState.Error;
    END_IF

  E_FanucHomingState.Done:
    // bDone is TRUE for one scan (derived below), then → Idle.
    stControl.Home := FALSE;
    _eState := E_FanucHomingState.Idle;

  E_FanucHomingState.Error:
    // bAt_Home did not go TRUE within tHomingTimeout.
    // Set bStart FALSE to reset.
    stControl.Home := FALSE;
    IF NOT bStart THEN
      _eState := E_FanucHomingState.Idle;
    END_IF

ELSE
  _eState := E_FanucHomingState.Error;

END_CASE

// ---------- Derived outputs ----------
eState := _eState;
bBusy  := (_eState = E_FanucHomingState.RequestHome) OR (_eState = E_FanucHomingState.WaitComplete);
bDone  := (_eState = E_FanucHomingState.Done);
bError := (_eState = E_FanucHomingState.Error);

END_FUNCTION_BLOCK

// POUs/FB_FanucOverwrite
// Writes a decimal value (0–nMax) to stControl.nDO3 (EtherCAT byte 3 / GI[25..33]).
// FB_FanucControl then writes the struct to aDO, so call this BEFORE fbControl.
FUNCTION_BLOCK FB_FanucOverwrite
VAR_INPUT
    nValue  : BYTE;          // Decimal value to send (0–nMax)
    bEnable : BOOL;           // TRUE = write nValue; FALSE = clear to 0
    nMax    : BYTE := 100;   // Upper limit — values above this set bError and write 0
END_VAR
VAR_IN_OUT
    stControl : ST_FanucControl;  // Control struct – wire same instance as FB_FanucEnable output
END_VAR
VAR_OUTPUT
    bError  : BOOL;   // TRUE if nValue exceeds nMax
    nActual : USINT;  // Value currently written
END_VAR

(*
  FB_FanucOverwrite
  Writes a decimal value to stControl.nDO3 (EtherCAT output byte 3 / GI[25..33]).
  FB_FanucControl maps the struct to aDO each scan, so this FB must be called
  BEFORE fbControl in MAIN — consistent with all other library FBs.

  TwinCAT maps the integer to 8 bits automatically. For example, value 5 (0000 0101)
  sets bits 0 and 2 on the FANUC GI channel; value 100 (0110 0100) sets bits 2, 5, 6.

  To extend the range beyond 100, increase nMax up to 255 (USINT limit).
*)

bError := nValue > nMax;

IF bEnable AND NOT bError THEN
    stControl.overwrite := nValue;
    nActual        := nValue;
ELSE
    stControl.overwrite := 0;
    nActual        := 0;
END_IF

END_FUNCTION_BLOCK

// POUs/FB_FanucStartProgram
//Starts a FANUC program in RSR mode (nProgram 1..8, one-hot 200 ms pulse), gated on bReady. bAck goes TRUE one scan when robot confirms start.
FUNCTION_BLOCK FB_FanucStartProgram
VAR_INPUT
  bStart   : BOOL;              // Rising edge: start program nProgram (gated on bReady)
  nProgram : INT;               // Program to start: 1..8 (RSR) or 1..255 (PNS)
  bReady   : BOOL;              // Gate: only start when robot is ready (FB_FanucEnable.bReady)
  stStatus : ST_FanucStatus;    // Live robot status – used for ACK feedback
END_VAR
VAR_IN_OUT
  stControl : ST_FanucControl;  // Modified in-place: Start_ProgramX 
END_VAR
VAR_OUTPUT
  bBusy  : BOOL;                      // TRUE while start pulse is active
  bDone  : BOOL;                      // One scan TRUE when pulse complete
  bAck   : BOOL;                      // One scan TRUE when robot acknowledges the start
  bError : BOOL;                      // TRUE if nProgram is out of range; set bStart FALSE to reset
  eState : E_FanucStartProgramState;  // Current state (diagnostic / HMI)
END_VAR
VAR
  _eState      : E_FanucStartProgramState := E_FanucStartProgramState.Idle;
  rtStart      : R_TRIG;  // Rising-edge detector on bStart AND bReady
  rtAck        : R_TRIG;  // Rising-edge detector for ACK feedback (RSR mode)
  rtPrgRunning : R_TRIG;  // Rising-edge detector for PROGRUN (PNS mode)
  tonPulse     : TON;     // 200 ms start pulse timer
  nActiveProg  : INT;     // Program number latched at trigger (stable during pulse)
END_VAR

(*
  FB_FanucStartProgram
  Triggers a FANUC robot program start in RSR mode.

  nProgram 1..8 maps to a one-hot 200 ms pulse on Start_Program1..8 (UI[9..16]).
  The robot acknowledges on the matching ACK bit (UO[11..18]); bAck goes TRUE for one scan.

  Usage:
    - Call every PLC cycle.
    - Pass the stControl struct that FB_FanucEnable populated (VAR_IN_OUT).
      This FB stamps only the Start_ProgramX bits; all other bits are preserved.
    - Wire bReady from FB_FanucEnable.bReady to gate starts.
    - Call FB_FanucControl AFTER this FB so it sees the final stControl state.

  Reset:
    bError latches if nProgram is out of range (1..8). Set bStart FALSE to reset.
*)

// --------- Edge detect ---------
rtStart(CLK := bStart AND bReady);

// --------- State machine ---------
CASE _eState OF

  E_FanucStartProgramState.Idle:
    stControl.Start_Program1 := FALSE;
    stControl.Start_Program2 := FALSE;
    stControl.Start_Program3 := FALSE;
    stControl.Start_Program4 := FALSE;
    stControl.Start_Program5 := FALSE;
    stControl.Start_Program6 := FALSE;
    stControl.Start_Program7 := FALSE;
    stControl.Start_Program8 := FALSE;
    tonPulse(IN := FALSE);
    IF rtStart.Q THEN
      IF nProgram < 1 OR nProgram > 8 THEN
        _eState := E_FanucStartProgramState.Error;
      ELSE
        nActiveProg := nProgram;
        _eState     := E_FanucStartProgramState.Pulsing;
      END_IF
    END_IF

  E_FanucStartProgramState.Pulsing:
    // One-hot: assert only the bit corresponding to nActiveProg for 200 ms.
    tonPulse(IN := TRUE, PT := T#200MS);
    CASE nActiveProg OF
      1: stControl.Start_Program1 := TRUE;
      2: stControl.Start_Program2 := TRUE;
      3: stControl.Start_Program3 := TRUE;
      4: stControl.Start_Program4 := TRUE;
      5: stControl.Start_Program5 := TRUE;
      6: stControl.Start_Program6 := TRUE;
      7: stControl.Start_Program7 := TRUE;
      8: stControl.Start_Program8 := TRUE;
    END_CASE
    IF tonPulse.Q THEN
      tonPulse(IN := FALSE);
      _eState := E_FanucStartProgramState.Done;
    END_IF

  E_FanucStartProgramState.Done:
    stControl.Start_Program1 := FALSE;
    stControl.Start_Program2 := FALSE;
    stControl.Start_Program3 := FALSE;
    stControl.Start_Program4 := FALSE;
    stControl.Start_Program5 := FALSE;
    stControl.Start_Program6 := FALSE;
    stControl.Start_Program7 := FALSE;
    stControl.Start_Program8 := FALSE;
    _eState := E_FanucStartProgramState.Idle;

  E_FanucStartProgramState.Error:
    stControl.Start_Program1 := FALSE;
    stControl.Start_Program2 := FALSE;
    stControl.Start_Program3 := FALSE;
    stControl.Start_Program4 := FALSE;
    stControl.Start_Program5 := FALSE;
    stControl.Start_Program6 := FALSE;
    stControl.Start_Program7 := FALSE;
    stControl.Start_Program8 := FALSE;
    IF NOT bStart THEN
      _eState := E_FanucStartProgramState.Idle;
    END_IF

ELSE
  _eState := E_FanucStartProgramState.Error;

END_CASE

// --------- ACK detection ---------
CASE nActiveProg OF
  1: rtAck(CLK := stStatus.bProg_Start1ACK);
  2: rtAck(CLK := stStatus.bProg_Start2ACK);
  3: rtAck(CLK := stStatus.bProg_Start3ACK);
  4: rtAck(CLK := stStatus.bProg_Start4ACK);
  5: rtAck(CLK := stStatus.bProg_Start5ACK);
  6: rtAck(CLK := stStatus.bProg_Start6ACK);
  7: rtAck(CLK := stStatus.bProg_Start7ACK);
  8: rtAck(CLK := stStatus.bProg_Start8ACK);
ELSE
  rtAck(CLK := FALSE);
END_CASE

// --------- Derived outputs ---------
eState := _eState;
bBusy  := (_eState = E_FanucStartProgramState.Pulsing);
bDone  := (_eState = E_FanucStartProgramState.Done);
bError := (_eState = E_FanucStartProgramState.Error);
bAck   := rtAck.Q;

END_FUNCTION_BLOCK
